FUNCTION_BLOCK PUBLIC Disposable_TestSuit EXTENDS TcUnit.FB_TestSuite
VAR
END_VAR

OnDisposeCalledFromDisposeMethod();
OnDisposeCalledByManuallyDeleting();
OnDisposeOnlyCalledOnceDuringCancel();
OnDisposeCalledWithExplicitFlagFalse();
OnDisposeCalledWithExplicitFlagTrue();

METHOD PUBLIC OnDisposeCalledByManuallyDeleting
VAR
	mockDispose : POINTER TO MockDisposable;
	disposed : BOOL;
END_VAR
TEST('OnDisposeCalledByManuallyDeleting');

// @TEST-FIXTURE
mockDispose := __NEW(MockDisposable(DisposedFlag:=disposed));

// @TEST-RUN
__DELETE(mockDispose);

// @TEST-ASSSERT
AssertTrue(
	Condition := disposed,
	Message := 'OnDispose was not correctly triggered in the MockDisposable'
);

TEST_FINISHED();
END_METHOD

METHOD PUBLIC OnDisposeCalledFromDisposeMethod
VAR
	mockDispose : POINTER TO MockDisposable;
	disposed : BOOL;
END_VAR
TEST('OnDisposeCalledFromDisposeMethod');

// @TEST-FIXTURE
mockDispose := __NEW(MockDisposable(DisposedFlag:=disposed));

// @TEST-RUN
mockDispose^.Dispose();

// @TEST-ASSSERT
AssertTrue(
	Condition := disposed,
	Message := 'OnDispose was not correctly triggered in the MockDisposable'
);

TEST_FINISHED();
END_METHOD

METHOD PUBLIC OnDisposeCalledWithExplicitFlagFalse
VAR
	mockDispose : POINTER TO MockDisposableWithExplicitFeedback;
	explicit : BOOL;
END_VAR
TEST('OnDisposeCalledWithExplicitFlagFalse');

// @TEST-FIXTURE
mockDispose := __NEW(MockDisposableWithExplicitFeedback(ExplicitFlag:=explicit));

// @TEST-RUN
__DELETE(mockDispose);

// @TEST-ASSSERT
AssertFalse(
	Condition := explicit,
	Message := 'OnDispose argument CalledExplicitly was not false when called implicitly'
);

TEST_FINISHED();
END_METHOD

METHOD PUBLIC OnDisposeCalledWithExplicitFlagTrue
VAR
	mockDispose : POINTER TO MockDisposableWithExplicitFeedback;
	explicit : BOOL;
END_VAR
TEST('OnDisposeCalledWithExplicitFlagTrue');

// @TEST-FIXTURE
mockDispose := __NEW(MockDisposableWithExplicitFeedback(ExplicitFlag:=explicit));

// @TEST-RUN
mockDispose^.Dispose();

// @TEST-ASSSERT
AssertTrue(
	Condition := explicit,
	Message := 'OnDispose argument CalledExplicitly was not true when called explicitly'
);

TEST_FINISHED();
END_METHOD

METHOD PUBLIC OnDisposeOnlyCalledOnceDuringCancel
VAR
	mockDispose : POINTER TO MockDisposableWithCancel;
	disposedCount : INT;
	expected : INT := 1;
END_VAR
TEST('OnDisposeOnlyCalledOnceDuringCancel');

// @TEST-FIXTURE
mockDispose := __NEW(MockDisposableWithCancel(DisposedCounterFlag:=disposedCount));

// @TEST-RUN
mockDispose^.Dispose(); // should trigger OnDisposed which will be cancelled;
mockDispose^.Dispose(); // should trigger __Delete

// @TEST-ASSSERT
AssertEquals(
	Expected := expected,
	Actual := disposedCount,
	Message := 'OnDispose was incorrectly triggered more than once following a cancel'
);

TEST_FINISHED();
END_METHOD

END_FUNCTION_BLOCK

(* stored: Version 1.1.0.1, ProductVersion 3.1.4024.12
   POU Disposable_TestSuit: Id {5e30d77d-5ab7-4a68-9932-9d53fc3729bd}, SpecialFunc None
   Method OnDisposeCalledByManuallyDeleting: Id {53f28239-f13a-41de-aa9f-47d3ff4c2a4d}
   Method OnDisposeCalledFromDisposeMethod: Id {f6d78085-e7eb-482f-b15d-638e7798de7e}
   Method OnDisposeCalledWithExplicitFlagFalse: Id {3a5dcb77-aaad-459c-8895-b710f6e010c5}
   Method OnDisposeCalledWithExplicitFlagTrue: Id {1c28e0a8-a446-43bb-8ecc-5edeb1700d70}
   Method OnDisposeOnlyCalledOnceDuringCancel: Id {20e38352-90f3-4ba0-9c2b-439ece13ab5d} *)
